Staubli VAL3: loadEditTraj.pgx

program loadEditTraj(string x_sName)
  local num i
begin
  // load the type
  call trajType:load(x_sName,i)
  if i!=0
    popUpMsg("Loading trajectory type "+x_sName+" error CODE "+toString("",i))
    logMsg("INTERFACE:TRAJECTORY LIBLOAD "+x_sName+" result "+toString("",i))
  endIf
end
